(* PLC project Unnamed, Unknown Unnamed 1 *)
(* stored: creationDateTime 2024-01-09T16:45:07, modificationDateTime 2024-01-23T14:31:54 *)

PROGRAM Add
  VAR_INPUT
    u1 : REAL;
    u2 : REAL;
  END_VAR
  VAR_OUTPUT
    y1 : REAL;
  END_VAR

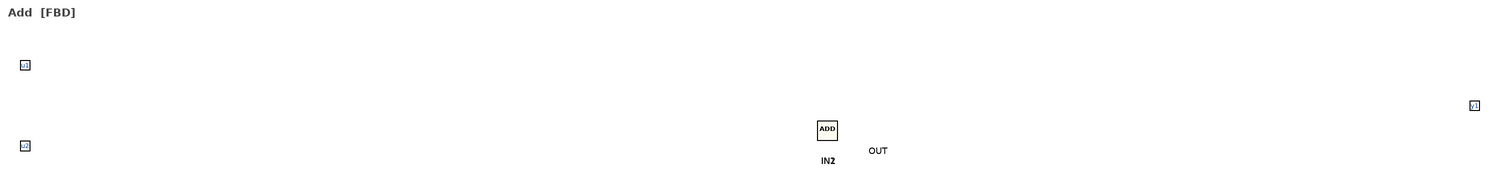
(* FBD diagram, written out as Structured Text *)
y1 := u1 + u2;
END_PROGRAM

CONFIGURATION config
  RESOURCE resource1 ON PLC
    TASK task0(INTERVAL := T#20ms, PRIORITY := 0);
    PROGRAM instance0 WITH task0 : Add;
  END_RESOURCE
END_CONFIGURATION
